// TwinCAT 3 PLC project LibrairieProject
// Title: Factorial
// Company: VibraSens
// Author: Antoine
// ProjectVersion: 1.0.0
// Description: Calcul le factoriel d'un nombre
// ProgramVersion: 3.1.4024.0
// libraries:
//   Tc2_Standard, * (Beckhoff Automation GmbH)
//   Tc2_System, * (Beckhoff Automation GmbH)
//   Tc3_Module, * (Beckhoff Automation GmbH)
// project tree:
//   POUs/ Factorial.TcPOU
//   Version/ Global_Version.TcGVL
// real-time tasks:
//   TASK PlcTask: cycle T#10ms, priority 20, ADS port 350

// ---- Version/Global_Version.TcGVL
{attribute 'TcGenerated'}
{attribute 'no-analysis'}
{attribute 'linkalways'}
// This function has been automatically generated from the project information.
VAR_GLOBAL CONSTANT
	{attribute 'const_non_replaced'}
	stLibVersion_Factorial : ST_LibVersion := (iMajor := 1, iMinor := 0, iBuild := 0, iRevision := 0, nFlags := 0, sVersion := '1.0.0');
END_VAR

// ---- POUs/Factorial.TcPOU
FUNCTION Factorial : ULINT
VAR_INPUT
	n : ULINT;
END_VAR
VAR
	nReturnValue : ULINT;
	i: ULINT;
END_VAR

nReturnValue := 1;
FOR i := 1 TO n BY 1 DO
	nReturnValue := nReturnValue * i;
END_FOR
Factorial := nReturnValue;

END_FUNCTION
